Fanuc KAREL source: kt00185.KL

-- PROVISIONAL review KL for V1013-1; original PC SHA256 533f9b96aabaa5e631cd11c5d393d345238f64a2574082bea6522bab4f683c5c
-- Incomplete behavior may be omitted. Consult companion uncertainty JSON. Do not deploy.
PROGRAM KT00185
%NOLOCKGROUP
VAR
  I2 : INTEGER
  OUT : INTEGER
-- UNRESOLVED_DECL H1 type=002017
BEGIN
  -- UNRESOLVED_PC offsets 5-19; opcodes 2E,22,9D,33,B4
  -- UNRESOLVED_PC offsets 24-35; opcodes 2E,23
  -- UNRESOLVED_PC offsets 40-62; opcodes 22,9D,33,B3,21,56,23
  -- UNRESOLVED_PC offsets 67-71; opcodes 7F
END KT00185
